// TIA Portal V18 export
FUNCTION "cab_main" : Void   // FC1, FBD
{ S7_Optimized_Access := 'TRUE' }
VERSION : 0.1
// stored: AutoNumber true, IsIECCheckEnabled false, SetENOAutomatically false, UDAEnableTagReadback false
   VAR_TEMP
      erCOM_A1 : Bool;
      wnDelay : Bool;
      er_нуевыеБлокировки : Bool;
      pt : Time;
   END_VAR
BEGIN

REGION Network 3
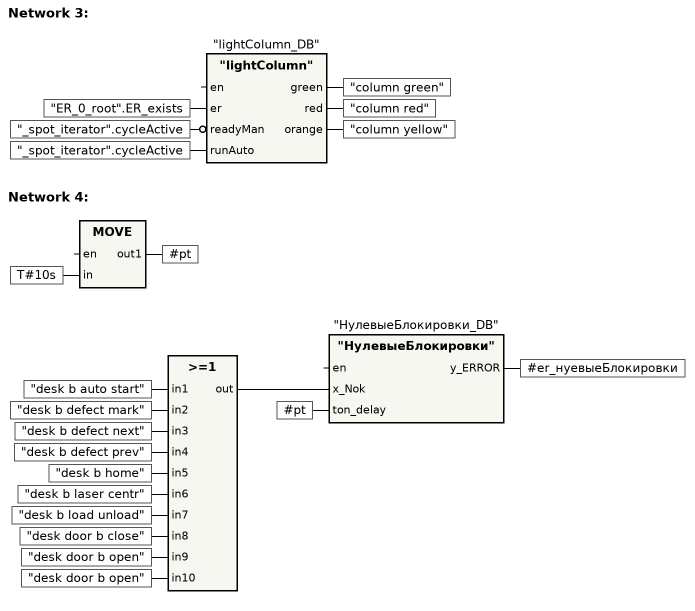
   "lightColumn_DB"(er := "ER_0_root".ER_exists,   // "lightColumn"
                    readyMan := NOT "_spot_iterator".cycleActive,
                    runAuto := "_spot_iterator".cycleActive,
                    green => "column green",
                    red => "column red",
                    orange => "column yellow");
END_REGION

REGION Network 4
   #pt := T#10s;
   "НулевыеБлокировки_DB"(x_Nok := "desk b auto start" OR "desk b defect mark" OR "desk b defect next" OR "desk b defect prev" OR "desk b home" OR "desk b laser centr" OR "desk b load unload" OR "desk door b close" OR "desk door b open" OR "desk door b open",   // "НулевыеБлокировки"
                          ton_delay := #pt,
                          y_ERROR => #er_нуевыеБлокировки);
END_REGION

REGION Network 5
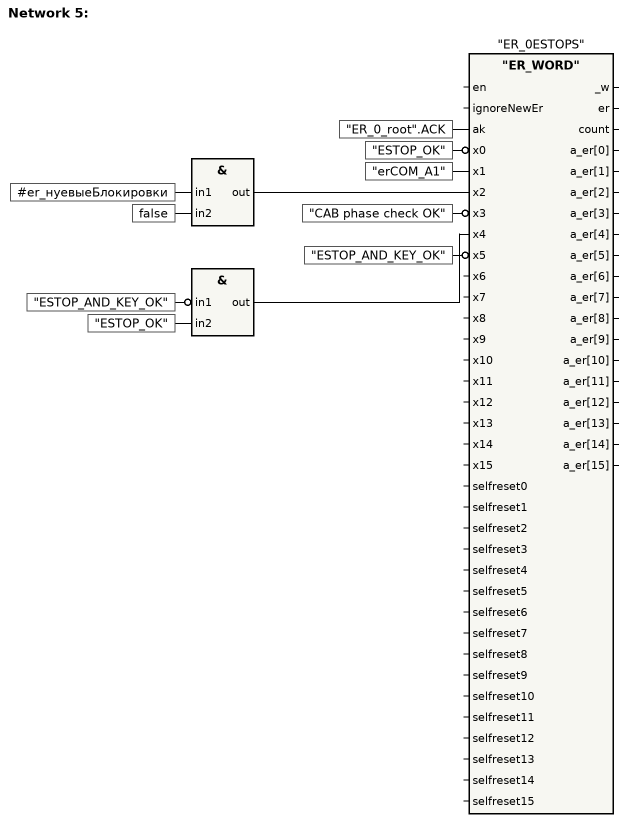
   "ER_0ESTOPS"(ak := "ER_0_root".ACK,   // "ER_WORD"
                x0 := NOT "ESTOP_OK",
                x1 := "erCOM_A1",
                x2 := #er_нуевыеБлокировки AND false,
                x3 := NOT "CAB phase check OK",
                x4 := NOT "ESTOP_AND_KEY_OK" AND "ESTOP_OK",
                x5 := NOT "ESTOP_AND_KEY_OK");
END_REGION

REGION Network 6
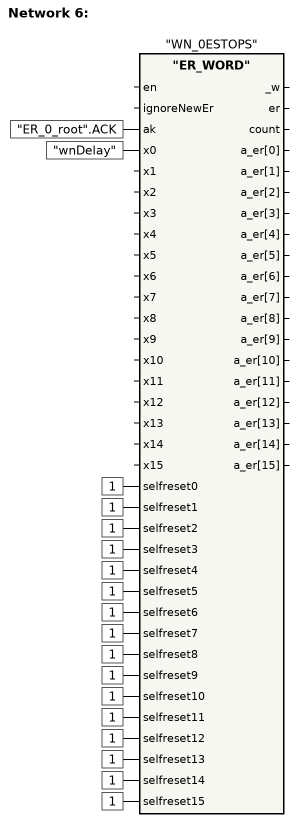
   "WN_0ESTOPS"(ak := "ER_0_root".ACK,   // "ER_WORD"
                x0 := "wnDelay",
                selfreset0 := 1,
                selfreset1 := 1,
                selfreset2 := 1,
                selfreset3 := 1,
                selfreset4 := 1,
                selfreset5 := 1,
                selfreset6 := 1,
                selfreset7 := 1,
                selfreset8 := 1,
                selfreset9 := 1,
                selfreset10 := 1,
                selfreset11 := 1,
                selfreset12 := 1,
                selfreset13 := 1,
                selfreset14 := 1,
                selfreset15 := 1);
END_REGION
END_FUNCTION
